// TIA Portal V20 export
// export: Created 2025-12-01T14:57:05.5007251Z, ExportSetting None, DisplayName Totally Integrated Automation Portal, DisplayVersion V20 Update 3, DisplayName TIA Portal Openness, DisplayVersion V20 Update 3, DisplayName TIA Portal Version Control Interface, DisplayVersion V20 Update 3, DisplayName STEP 7 Professional, DisplayVersion V20 Update 3, DisplayName STEP 7 Safety, DisplayVersion V20 Update 2, DisplayName WinCC Basic/Comfort/Advanced, DisplayVersion V20 Update 3, DisplayName WinCC Professional, DisplayVersion V20 Update 3, DisplayName WinCC Unified, DisplayVersion V20 Update 3
FUNCTION "FC896_LeerZonaMemoria" : Void   // FC896, LAD
TITLE = "LeerZonaMemoria" - Escribir en la String una Zona de Memoria
{ S7_Optimized_Access := 'FALSE' }
AUTHOR : TRACKING
NAME : 20130301
VERSION : 3.0
// stored: AutoNumber false, SetENOAutomatically false
   VAR_INPUT
      DB_String : UInt;   // Numero de DB del String
      OffsetIni : UInt;   // Numero de Byte de Inicio de la String
      TipoMemoria : UInt;   // Tipo de Memoria a Leer
      NumeroMemoria : UInt;   // Numero de Memoria a Leer
      OffsetMemoria : UInt;   // Offset de la Memoria a Leer
      LongitudMemoria : UInt;   // Longitud de la Memoria a Leer
   END_VAR
   VAR_OUTPUT
      OffsetFin : UInt;   // Numero de Byte Final de la String
   END_VAR
   VAR_TEMP
      NumDBOrigen : Word;   // Num. de DB de Origen
      NumDBDestino : Word;   // Num. de DB de Destino
      P_Origen : DWord;   // Puntero al Origen
      P_Destino : DWord;   // Puntero al Destino
      ContadorBytes : UInt;   // Numero de Bytes Traspasados
      ByteLeido : Byte;   // Byte leido de la Memoria
      ByteBaja : Byte;   // Parte Baja del Byte leido de la Memoria
      ByteAlta : Byte;   // Parte Alta del Byte leido de la Memoria
   END_VAR
BEGIN

NETWORK
TITLE = Inicializaciones
// - Inicializar diferentaes Variables
// ---------------------------------------------------------------------------
// --- Variables internas

      L     #OffsetIni;  // Ini. Devolucion de la Función
      T     #OffsetFin;

// ---------------------------------------------------------------------------
// --- Variables de Origen y destino

      L     #DB_String;  // Variables de Destino
      T     #NumDBDestino;
      L     #OffsetIni;
      SLD   3;
      T     #P_Destino;  // Puntero a la String

      L     #NumeroMemoria;  // Variables de Origen
      T     #NumDBOrigen;
      L     #OffsetMemoria;
      SLD   3;
      T     #P_Origen;  // Puntero a la Zona Memoria


NETWORK
TITLE = Realizar la transferencia
// Bucle de Lectura de la zona de Memoria
// ---------------------------------------------------------------------------
// --- Bucle para la Trasferencia

      L     0;
      T     #ContadorBytes;  // Inicializa el Contador

C_BU: L     #ContadorBytes;
      L     #LongitudMemoria;
      ==I;
      JC    _END;  // Se ha transferido todos ?

      L     #P_Origen;
      LAR1;
      OPN   DB [#NumDBOrigen];
      L     DBB [AR1, P#0.0];  // Leer el siguiente Byte de Memoria
      T     #ByteLeido;
      +AR1  P#1.0;
      T     #P_Origen;

      JU    CV_B;  // Ir a Convertirlo a ASCII



NETWORK
TITLE = Conversion del Byte de Memoria
// Realizando la conversion de un Byte HEX -> un Word en ASCII
// ---------------------------------------------------------------------------
// --- Leer la Parte Baja del Byte y Convertir el ASCII

CV_B: L     #ByteLeido;  // Recoger la Parte Baja del Byte
      L     W#16#F;
      AW;
      T     #ByteBaja;

      L     #ByteBaja;  // Mirar si es Letra o Numero
      L     9;
      >I;
      JC    BB_L;

      L     #ByteBaja;  // Es Numero -> Convertir a ASCII
      L     W#16#30;
      +I;
      T     #ByteBaja;

      JU    CV_A;  // Ir a Conversion de la Parte Alta

BB_L: L     #ByteBaja;  // Es Letra -> Convertir a ASCII
      L     W#16#37;
      +I;
      T     #ByteBaja;

      JU    CV_A;  // Ir a Conversion de la Parte Alta

// ---------------------------------------------------------------------------
// --- Leer la Parte Alta del Byte y Convertir el ASCII

CV_A: L     #ByteLeido;  // Recoger la Parte Alta del Byte
      L     W#16#F0;
      AW;
      SRD   4;
      L     #ByteAlta;

      L     #ByteAlta;  // Mirar si es Letra o Numero
      L     9;
      >I;
      JC    BA_L;

      L     #ByteAlta;  // Es Numero -> Convertir a ASCII
      L     W#16#30;
      +I;
      T     #ByteAlta;

      JU    CV_F;  // Ir a Final de Conversion

BA_L: L     #ByteAlta;  // Es Letra -> Convertir a ASCII
      L     W#16#37;
      +I;
      T     #ByteAlta;

      JU    CV_F;  // Ir a Final de Conversion

// ---------------------------------------------------------------------------
// --- Final de la Convertidor del Byte a Word

CV_F: L     #P_Destino;  // Traspasar a String
      LAR1;
      OPN   DB [#NumDBDestino];
      L     #ByteAlta;
      T     DBB [AR1, P#0.0];  // Parte Alta -> String
      L     #ByteBaja;
      T     DBB [AR1, P#1.0];  // Parte Baja -> String
      +AR1  P#2.0;
      T     #P_Destino;

      L     #ContadorBytes;  // Leido un Byte mas de la Memoria
      L     1;
      +I;
      T     #ContadorBytes;

      JU    C_BU;


NETWORK
TITLE = Final
// Se Acabo la funcion
_END: L     #P_Destino;
      SRD   3;
      T     #OffsetFin;  // Numero de Bytes que tiene


END_FUNCTION
